PROGRAM MAIN
VAR
END_VAR

PB_Initialisation();
PB_ObjectExecution();

END_PROGRAM

(* stored: Version 1.1.0.1, ProductVersion 3.1.4024.9
   POU MAIN: Id {0e846b38-986c-4df4-8c71-58119a6eaca3}, SpecialFunc None *)
